Omron CX-Programmer project NuevoProyecto (CX-Programmer 9.61)

# PLC NuevoPLC1: CJ2M CPU11

## Program NuevoPrograma1 (cyclic task 0)
Local symbols
BVerde 0.00 BOOL
B_Mas 1.01 BOOL
B_Menos 1.02 BOOL
C_Mas 1.03 BOOL
C_Menos 1.04 BOOL
CilindroE_ON 1.06 BOOL
D_Mas 1.05 BOOL
E_0 2.00 BOOL
E_1 2.01 BOOL
E_2 2.02 BOOL
E_3 2.03 BOOL
E_4 2.04 BOOL
E_5 2.05 BOOL
E_6 2.06 BOOL
E_7 2.07 BOOL
E_8 2.08 BOOL
E_9 2.09 BOOL
I2P1 0.02 BOOL
I3PD 0.04 BOOL
I3PI 0.03 BOOL
b_mas 0.07 BOOL
b_menos 0.08 BOOL
c_mas 0.09 BOOL
c_meno 0.12 BOOL
c_menos 0.10 BOOL
d_mas 0.11 BOOL

### Section main
; rung 0
; cells of this rung as drawn
  row 0 col 0: LD E_8
  row 0 col 6: OUT E_9
  vertical links (row, left of col): 
; rung 1
; cells of this rung as drawn
  row 0 col 6: OUT E_8
  vertical links (row, left of col): 

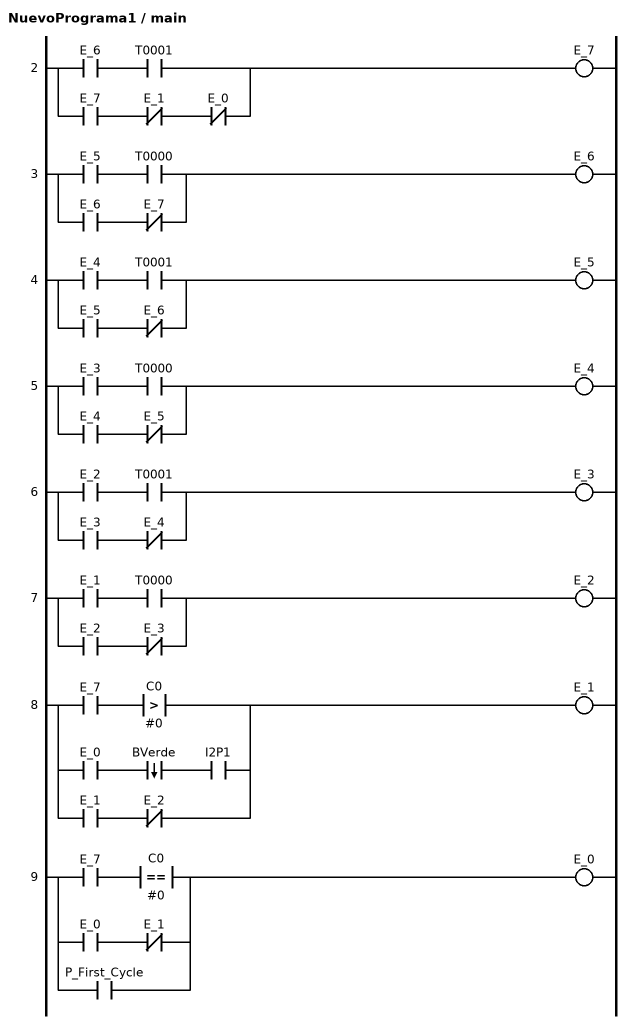
; rung 2
LD E_6
AND T0001
LD E_7
ANDNOT E_1
ANDNOT E_0
ORLD
OUT E_7
; rung 3
LD E_5
AND T0000
LD E_6
ANDNOT E_7
ORLD
OUT E_6
; rung 4
LD E_4
AND T0001
LD E_5
ANDNOT E_6
ORLD
OUT E_5
; rung 5
LD E_3
AND T0000
LD E_4
ANDNOT E_5
ORLD
OUT E_4
; rung 6
LD E_2
AND T0001
LD E_3
ANDNOT E_4
ORLD
OUT E_3
; rung 7
LD E_1
AND T0000
LD E_2
ANDNOT E_3
ORLD
OUT E_2
; rung 8
LD E_7
AND>(320) C0 #0
LD E_0
%AND BVerde
AND I2P1
ORLD
LD E_1
ANDNOT E_2
ORLD
OUT E_1
; rung 9
LD E_7
AND=(300) C0 #0
LD E_0
ANDNOT E_1
ORLD
OR P_First_Cycle
OUT E_0

### Section Salidas

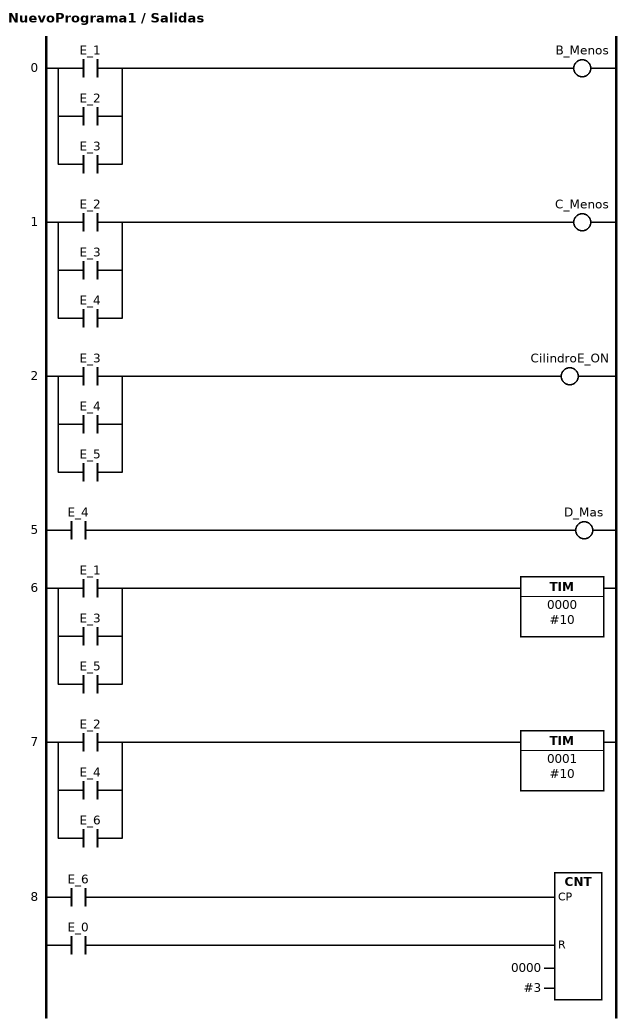
; rung 0
LD E_1
OR E_2
OR E_3
OUT B_Menos
; rung 1
LD E_2
OR E_3
OR E_4
OUT C_Menos
; rung 2
LD E_3
OR E_4
OR E_5
OUT CilindroE_ON
; rung 3
; cells of this rung as drawn
  row 0 col 6: OUT B_Mas
  vertical links (row, left of col): 
; rung 4
; cells of this rung as drawn
  row 0 col 6: OUT C_Mas
  vertical links (row, left of col): 
; rung 5
LD E_4
OUT D_Mas
; rung 6
LD E_1
OR E_3
OR E_5
TIM 0000 #10
; rung 7
LD E_2
OR E_4
OR E_6
TIM 0001 #10
; rung 8
LD E_6
LD E_0
CNT 0000 #3

### Section END
; rung 0
END(001)